(********************* G.D S.p.A. - Technical Department ***********************************
This program has been generated automatically from Application Designer DE&F
********************************************************************************************)
PROGRAM dbg_csp_case_main_services
VAR
  reset_output_test_shd : digital_output_shadow;
END_VAR

_objects_manager();

IF	g_application_status <> APPLICATION_STATUS_RUNNING
THEN
	RETURN;
END_IF

CASE process_get_mode(CONVERSION_this := dbg_root.prc) OF
	MODE_ABSENT,
	MODE_INACTIVE:
		RETURN;
	MODE_TEST:
		RETURN;
END_CASE

ACTION _objects_manager:
IF	objects_initialization()
THEN
	digital_output_shadow_init(
		sim_mode:= SHADOW_SIMULATION_MODE_AUTOMATIC, 
		father:= csp_case_main_services.reset_output_test, 
		process:= dbg_root.prc, 
		CONVERSION_this:= reset_output_test_shd);

	RETURN;
END_IF

IF	objects_running()
THEN
	digital_output_shadow_cycle(reset_output_test_shd);
END_IF
END_ACTION

END_PROGRAM

(* stored: Version 1.1.0.1, ProductVersion 3.1.4022.12
   POU dbg_csp_case_main_services: Id {65099fd7-1dad-434a-a7e6-0fb90607e357}, SpecialFunc None
   Action _objects_manager: Id {827bed1c-1720-4817-9880-f9419dcee906} *)
